FUNCTION_BLOCK L4_FMS205_F6Prueba_SFC EXTENDS L1_ControllerBase_SFC

VAR_IN_OUT
	Alime			: L3_Alimentador;
	Carga		 	: L3_PickAndPlace;
	Medid			: L3_MedidorTapa;
	Induc		 	: L3_CaptadorInductivo;
	Fotoe			: L3_DetectorFotoelectrico;
	Evacu		 	: L3_Evacuador;
	Desca			: L3_PickAndPlace;
	Plato			: L3_PlatoDivisor;
	Cinta			: L3_Cinta;
END_VAR

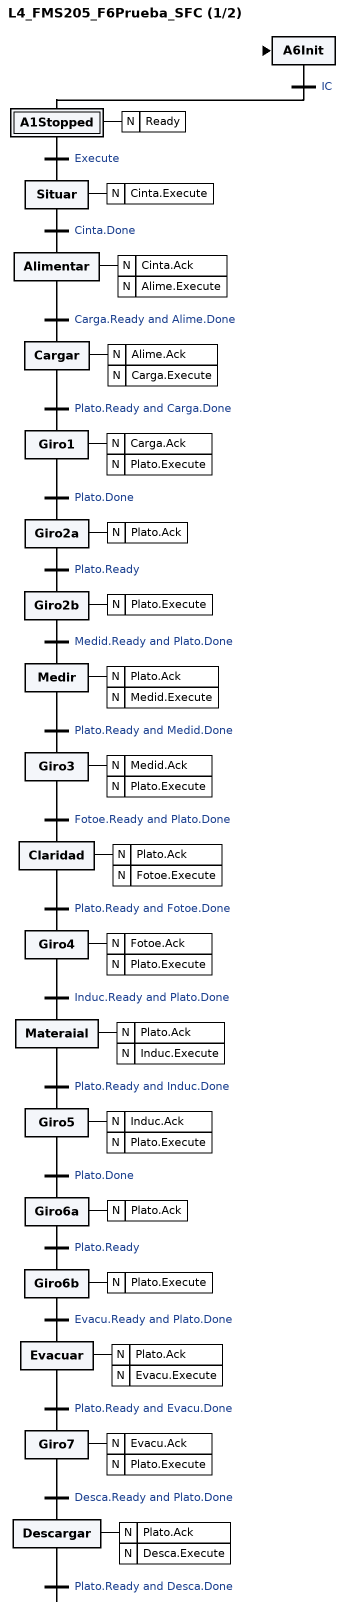
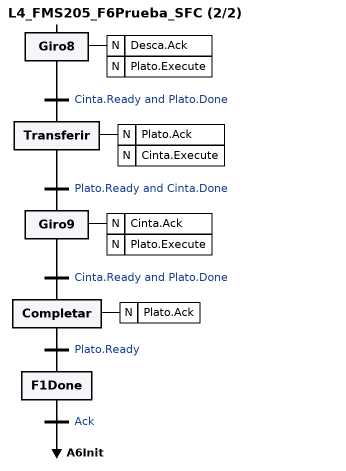
STEP A6Init:
END_STEP
TRANSITION FROM A6Init TO A1Stopped
    := IC;
END_TRANSITION
INITIAL_STEP A1Stopped:
    Ready(N);
END_STEP
TRANSITION FROM A1Stopped TO Situar
    := Execute;
END_TRANSITION
STEP Situar:
    Cinta.Execute(N);
END_STEP
TRANSITION FROM Situar TO Alimentar
    := Cinta.Done;
END_TRANSITION
STEP Alimentar:
    Cinta.Ack(N);
    Alime.Execute(N);
END_STEP
TRANSITION FROM Alimentar TO Cargar
    := Carga.Ready and Alime.Done;
END_TRANSITION
STEP Cargar:
    Alime.Ack(N);
    Carga.Execute(N);
END_STEP
TRANSITION FROM Cargar TO Giro1
    := Plato.Ready and Carga.Done;
END_TRANSITION
STEP Giro1:
    Carga.Ack(N);
    Plato.Execute(N);
END_STEP
TRANSITION FROM Giro1 TO Giro2a
    := Plato.Done;
END_TRANSITION
STEP Giro2a:
    Plato.Ack(N);
END_STEP
TRANSITION FROM Giro2a TO Giro2b
    := Plato.Ready;
END_TRANSITION
STEP Giro2b:
    Plato.Execute(N);
END_STEP
TRANSITION FROM Giro2b TO Medir
    := Medid.Ready and Plato.Done;
END_TRANSITION
STEP Medir:
    Plato.Ack(N);
    Medid.Execute(N);
END_STEP
TRANSITION FROM Medir TO Giro3
    := Plato.Ready and Medid.Done;
END_TRANSITION
STEP Giro3:
    Medid.Ack(N);
    Plato.Execute(N);
END_STEP
TRANSITION FROM Giro3 TO Claridad
    := Fotoe.Ready and Plato.Done;
END_TRANSITION
STEP Claridad:
    Plato.Ack(N);
    Fotoe.Execute(N);
END_STEP
TRANSITION FROM Claridad TO Giro4
    := Plato.Ready and Fotoe.Done;
END_TRANSITION
STEP Giro4:
    Fotoe.Ack(N);
    Plato.Execute(N);
END_STEP
TRANSITION FROM Giro4 TO Materaial
    := Induc.Ready and Plato.Done;
END_TRANSITION
STEP Materaial:
    Plato.Ack(N);
    Induc.Execute(N);
END_STEP
TRANSITION FROM Materaial TO Giro5
    := Plato.Ready and Induc.Done;
END_TRANSITION
STEP Giro5:
    Induc.Ack(N);
    Plato.Execute(N);
END_STEP
TRANSITION FROM Giro5 TO Giro6a
    := Plato.Done;
END_TRANSITION
STEP Giro6a:
    Plato.Ack(N);
END_STEP
TRANSITION FROM Giro6a TO Giro6b
    := Plato.Ready;
END_TRANSITION
STEP Giro6b:
    Plato.Execute(N);
END_STEP
TRANSITION FROM Giro6b TO Evacuar
    := Evacu.Ready and Plato.Done;
END_TRANSITION
STEP Evacuar:
    Plato.Ack(N);
    Evacu.Execute(N);
END_STEP
TRANSITION FROM Evacuar TO Giro7
    := Plato.Ready and Evacu.Done;
END_TRANSITION
STEP Giro7:
    Evacu.Ack(N);
    Plato.Execute(N);
END_STEP
TRANSITION FROM Giro7 TO Descargar
    := Desca.Ready and Plato.Done;
END_TRANSITION
STEP Descargar:
    Plato.Ack(N);
    Desca.Execute(N);
END_STEP
TRANSITION FROM Descargar TO Giro8
    := Plato.Ready and Desca.Done;
END_TRANSITION
STEP Giro8:
    Desca.Ack(N);
    Plato.Execute(N);
END_STEP
TRANSITION FROM Giro8 TO Transferir
    := Cinta.Ready and Plato.Done;
END_TRANSITION
STEP Transferir:
    Plato.Ack(N);
    Cinta.Execute(N);
END_STEP
TRANSITION FROM Transferir TO Giro9
    := Plato.Ready and Cinta.Done;
END_TRANSITION
STEP Giro9:
    Cinta.Ack(N);
    Plato.Execute(N);
END_STEP
TRANSITION FROM Giro9 TO Completar
    := Cinta.Ready and Plato.Done;
END_TRANSITION
STEP Completar:
    Plato.Ack(N);
END_STEP
TRANSITION FROM Completar TO F1Done
    := Plato.Ready;
END_TRANSITION
STEP F1Done:
END_STEP
TRANSITION FROM F1Done TO A6Init
    := Ack;
END_TRANSITION

END_FUNCTION_BLOCK

(* stored: Version 1.1.0.1, ProductVersion 3.1.4024.11
   POU L4_FMS205_F6Prueba_SFC: Id {a81c472c-1220-4b76-860b-f7f6b111694f}, SpecialFunc None *)
